(*~
	<docu>
		<summary>
			Describes the step status inside the sequencer.
		</summary>				
	</docu>	
~*)
{attribute 'qualified_only'}
{attribute 'strict'}
TYPE eStepStatus :
(
(*~
	<docu>
		<summary>
			No status defined.
		</summary>				
	</docu>	
~*)	
	None := 0,
(*~
	<docu>
		<summary>
			Step is disabled and it is not going to be executed.
			Next enabled step in the sequence will be executed, when sequencer reach that step.
		</summary>				
	</docu>	
~*)	
	Disabled := 10,
(*~
	<docu>
		<summary>
			Step is ready to run. This case occurs when sequence is in step mode, step is in order of the execution and step is enabled.
			Code body of the current step is not executing. After calling StepIn method, step becames running and its code body starts to be executing.
		</summary>				
	</docu>	
~*)	
	ReadyToRun := 20,
(*~
	<docu>
		<summary>
			Step is currently running and his code body is currently executing.
		</summary>				
	</docu>	
~*)	
	Running := 30,	
(*~
	<docu>
		<summary>
			Step has been finished. Its code body is not executing.
		</summary>				
	</docu>	
~*)	
	Done := 40,
(*~
	<docu>
		<summary>
			Step is in error state. Its code body is not executing.
		</summary>				
	</docu>	
~*)	
	Error := 50
);
END_TYPE

(* stored: Version 1.1.0.1, ProductVersion 3.1.4024.6
   DUT eStepStatus: Id {06e3f1be-90df-4a49-be95-caa6a15c597d} *)
